// TIA Portal V20 export
// export: Created 2025-12-01T14:57:11.4895268Z, ExportSetting None, DisplayName Totally Integrated Automation Portal, DisplayVersion V20 Update 3, DisplayName TIA Portal Openness, DisplayVersion V20 Update 3, DisplayName TIA Portal Version Control Interface, DisplayVersion V20 Update 3, DisplayName STEP 7 Professional, DisplayVersion V20 Update 3, DisplayName STEP 7 Safety, DisplayVersion V20 Update 2, DisplayName WinCC Basic/Comfort/Advanced, DisplayVersion V20 Update 3, DisplayName WinCC Professional, DisplayVersion V20 Update 3, DisplayName WinCC Unified, DisplayVersion V20 Update 3
FUNCTION "FC741_GestorDispositivoCBOX" : Void   // FC741, LAD
{ S7_Optimized_Access := 'FALSE' }
// stored: AutoNumber false, SetENOAutomatically false
   VAR_INPUT
      NumCBOX : UInt;   // Numero de VTDC a Gestionar
   END_VAR
   VAR_TEMP
      RecProtocoloDispositivo : "UDT_ProtocoloRecDispositivo";   // Protocolo De Ordenes
      EmiProtocoloDispositivo : "UDT_ProtocoloEmiDispositivo";   // Protocolo De Emisiones
      P_RecProtocolo : DWord;   // Puntero a la Variable Rec Protocolo
      P_EmiProtocolo : DWord;   // Puntero a la Variable Emi Protocolo
      P_Eventos : DWord;   // Eventos - Puntero al DB de Eventos
      DBEventos : Word;   // Eventos - DB de Eventos
      NumDBEventos : UInt;   // Eventos - DB de Eventos
      MaxBytesDeEventos : UInt;   // Eventos - Maximo Bytes en el DB de Eventos
      NumBytes : UInt;   // Eventos - Numero de Bytes en el DB de Eventos
      Conversion : DWord;   // Eventos - Valor Etiqueta Convertido
      Valor : UDInt;   // Eventos - Valor Numerico a Convertir
      Convertir : UInt;   // Eventos - Valor Etiqueta a Convertir
      OffsetFinal : UInt;   // Eventos - Posicion Final
      OffsetInicial : UInt;   // Eventos - Posicion Inicial
      NumeroDispositivo : UInt;   // Temporal - Numero de CBOX
      P_Temporal : DWord;   // Temporal - Puntero
   END_VAR
BEGIN

NETWORK
TITLE = Inicializar
////////////////////////////////////////////////////////////////////////////////////////
////////////////////////////////////////////////////////////////////////////////////////
////////////////////////////////////////////////////////////////////////////////////////
// --- Inicializar Variables

      L     #NumCBOX;
      T     #NumeroDispositivo;


////////////////////////////////////////////////////////////////////////////////////////
////////////////////////////////////////////////////////////////////////////////////////
////////////////////////////////////////////////////////////////////////////////////////
// --- Recoger Protocolo de ORDEN del Dispositivo
      CALL  MOVE
      ( IN  := "DB841_Recepcion".DispoArmario[#NumeroDispositivo].Protocolo,
        OUT := #RecProtocoloDispositivo
      );

      L     P##RecProtocoloDispositivo;
      T     #P_RecProtocolo;

////////////////////////////////////////////////////////////////////////////////////////
////////////////////////////////////////////////////////////////////////////////////////
////////////////////////////////////////////////////////////////////////////////////////
// --- Recoger Protocolo de EMISION del Dispositivo
      CALL  MOVE
      ( IN  := "DB840_Emision".DispoArmario[#NumeroDispositivo].Protocolo,
        OUT := #EmiProtocoloDispositivo
      );

      L     P##EmiProtocoloDispositivo;
      T     #P_EmiProtocolo;

      L     "DB840_Emision".DispoArmario[#NumeroDispositivo].Error;
      T     "DB830_Dispositivos".Dispositivos[#NumeroDispositivo].ErrorReal;

      L     LW [#P_EmiProtocolo];
      L     W#16#7700;  // Solo la Parte Baja
      AW;
      SRD   8;
      T     "DB830_Dispositivos".Dispositivos[#NumeroDispositivo].StatusReal;



NETWORK
TITLE = Generacion de Ordenes
GeneradorDeOrdenes:NOP   0;

////////////////////////////////////////////////////////////////////////////////////////
////////////////////////////////////////////////////////////////////////////////////////
////////////////////////////////////////////////////////////////////////////////////////
// --- Fase 01 : Cierre de Protocolo de la ORDEN
      L     "DB830_Dispositivos".Dispositivos[#NumeroDispositivo].EstadoOrdenDispo;
      L     0;
      <>I;  // Mirar si no esta Cerrado el Protocolo ?
      JC    Cerrar_ProtocoloOrdenes;


////////////////////////////////////////////////////////////////////////////////////////
////////////////////////////////////////////////////////////////////////////////////////
////////////////////////////////////////////////////////////////////////////////////////
// --- Fase 02 : Eventos Recibidos (Distribucion)
      L     "DB830_Dispositivos".Dispositivos[#NumeroDispositivo].EstadoRecepcionEvento;
      L     0;  // Se han Recibido Eventos
      ==I;
      JC    Final_GeneradorDeOrdenes;


////////////////////////////////////////////////////////////////////////////////////////
// --- (260) Cambio de Estado sin Orden
      SET;
      SET;
      L     "DB830_Dispositivos".Dispositivos[#NumeroDispositivo].EstadoRecepcionEvento;
      L     260;
      ==I;
      JC    EventoRecibido_PeticionRefrescoDatos;


////////////////////////////////////////////////////////////////////////////////////////
// --- (261...274) - Recibido Ordenes para el Dispositivo
      SET;
      A(;
      L     "DB830_Dispositivos".Dispositivos[#NumeroDispositivo].EstadoRecepcionEvento;
      L     "Evento_DISPOSITIVO_InicioOrdenDipositivo";
      >=I;
      );
      A(;
      L     "DB830_Dispositivos".Dispositivos[#NumeroDispositivo].EstadoRecepcionEvento;
      L     "Evento_DISPOSITIVO_FinalOrdenDispositivo";
      <=I;
      );
      JC    EventoRecibido_OrdenesDelDipositivo;


////////////////////////////////////////////////////////////////////////////////////////
// --- (250) Peticion de Refesco de Datos del Dispositivo
      SET;
      L     "DB830_Dispositivos".Dispositivos[#NumeroDispositivo].EstadoRecepcionEvento;
      L     "Evento_DISPOSITIVO_PeticionEstadoActual";
      ==I;
      JC    EventoRecibido_PeticionRefrescoDatos;


////////////////////////////////////////////////////////////////////////////////////////
// --- No existe este Evento Programado
      L     0;  // Eliminar Evento
      T     "DB830_Dispositivos".Dispositivos[#NumeroDispositivo].EstadoRecepcionEvento;


////////////////////////////////////////////////////////////////////////////////////////
////////////////////////////////////////////////////////////////////////////////////////
////////////////////////////////////////////////////////////////////////////////////////
// --- Fase Final - No hay que hacer mas en la Generacion de Ordenes
//                  Seguir con el Generador de Emisiones
Final_GeneradorDeOrdenes:NOP   0;
      JU    GeneradorDeEmisiones;



NETWORK
TITLE = ---- Cierre del Protocolo de Ordenes del Dispositivo
Cerrar_ProtocoloOrdenes:NOP   0;

////////////////////////////////////////////////////////////////////////////////////////
////////////////////////////////////////////////////////////////////////////////////////
////////////////////////////////////////////////////////////////////////////////////////
// --- Distribuir dependiendo de la Fase del Protocolo de ORDEN

      L     "DB830_Dispositivos".Dispositivos[#NumeroDispositivo].EstadoOrdenDispo;
      L     1;
      ==I;
      JC    EnFase_01_ProtocoloOrdenes;
      JU    EnFase_02_ProtocoloOrdenes;


////////////////////////////////////////////////////////////////////////////////////////
////////////////////////////////////////////////////////////////////////////////////////
////////////////////////////////////////////////////////////////////////////////////////
// --- En Fase 01 : Esperando que se Desactive RecepOK del Dispositivo
EnFase_01_ProtocoloOrdenes:NOP   0;
      SET;  // DesActivado la RecepOK ?
      A     "DB840_Emision".DispoArmario[#NumeroDispositivo].Protocolo.RecepOK;
      JC    FinCierre_ProtocoloOrdenes;

// --- Finalizado el Protocolo
      L     0;
      T     "DB830_Dispositivos".Dispositivos[#NumeroDispositivo].EstadoOrdenDispo;
      JU    FinCierre_ProtocoloOrdenes;


////////////////////////////////////////////////////////////////////////////////////////
////////////////////////////////////////////////////////////////////////////////////////
////////////////////////////////////////////////////////////////////////////////////////
// --- Esperando que se active RecepOK del Dispositivo
EnFase_02_ProtocoloOrdenes:NOP   0;
      SET;  // DesActivado la RecepOK ?
      AN    "DB840_Emision".DispoArmario[#NumeroDispositivo].Protocolo.RecepOK;
      JC    FinCierre_ProtocoloOrdenes;

// --- Fase 01 del Protocolo
      L     1;
      T     "DB830_Dispositivos".Dispositivos[#NumeroDispositivo].EstadoOrdenDispo;

      L     LW [#P_RecProtocolo];
      L     W#16#80;
      AW;  // Desactivo la Orden enviada
      T     LW [#P_RecProtocolo];

      CALL  MOVE
      ( IN  := #RecProtocoloDispositivo,
        OUT := "DB841_Recepcion".DispoArmario[#NumeroDispositivo].Protocolo
      );

      L     0;  // Borrar Variables Auxiliares
      T     "DB841_Recepcion".DispoArmario[#NumeroDispositivo].Auxiliar_01;
      T     "DB841_Recepcion".DispoArmario[#NumeroDispositivo].Auxiliar_02;
      T     "DB841_Recepcion".DispoArmario[#NumeroDispositivo].Auxiliar_03;
      T     "DB841_Recepcion".DispoArmario[#NumeroDispositivo].ORDE;

      JU    FinCierre_ProtocoloOrdenes;


////////////////////////////////////////////////////////////////////////////////////////
////////////////////////////////////////////////////////////////////////////////////////
////////////////////////////////////////////////////////////////////////////////////////
FinCierre_ProtocoloOrdenes:NOP   0;
      JU    Final_GeneradorDeOrdenes;



NETWORK
TITLE = ---- (261...274) Recibido Ordenes para el Dipositivo
EventoRecibido_OrdenesDelDipositivo:NOP   0;

////////////////////////////////////////////////////////////////////////////////////////
////////////////////////////////////////////////////////////////////////////////////////
////////////////////////////////////////////////////////////////////////////////////////
// --- (261...274) Recibido Ordenes para el Dipositivo
      L     "DB830_Dispositivos".Dispositivos[#NumeroDispositivo].EstadoRecepcionEvento;
      L     260;
      -I;  // Numero de Bit a Activar
      L     #P_RecProtocolo;
      +D;  // Direccion del Bit a Activar
      T     #P_Temporal;

////////////////////////////////////////////////////////////////////////////////////////
// --- Activar Orden Recibida (Nuevo Estado)

      SET;  // Poner a '1' el bit de la orden
      S     L [#P_Temporal];  // Orden del PLC calculada

      CALL  MOVE
      ( IN  := #RecProtocoloDispositivo,
        OUT := "DB841_Recepcion".DispoArmario[#NumeroDispositivo].Protocolo
      );


////////////////////////////////////////////////////////////////////////////////////////
// --- Darlo por tratado y Activar Protocolo
      L     2;  // Fase 2 - Esperando que active el RecepOK
      T     "DB830_Dispositivos".Dispositivos[#NumeroDispositivo].EstadoOrdenDispo;
      L     0;  // Darlo por tratado
      T     "DB830_Dispositivos".Dispositivos[#NumeroDispositivo].EstadoRecepcionEvento;


////////////////////////////////////////////////////////////////////////////////////////
// --- Final del Evento
      JU    Final_GeneradorDeOrdenes;



NETWORK
TITLE = ---- (250 ) Peticion de Refresco de Datos del Dispositivo
EventoRecibido_PeticionRefrescoDatos:NOP   0;

////////////////////////////////////////////////////////////////////////////////////////
////////////////////////////////////////////////////////////////////////////////////////
////////////////////////////////////////////////////////////////////////////////////////
// --- 250 -  Recibido Evento de Refresco de Datos para el Dispositivo
      L     "DB830_Dispositivos".Dispositivos[#NumeroDispositivo].EstadoEmisionEvento;
      L     0;
      <>I;
      JC    Final_GeneradorDeOrdenes;


// --- (160) Refresco de datos del dispositivo
      L     "Evento_DISPOSITIVO_EstadoActual";
      T     "DB830_Dispositivos".Dispositivos[#NumeroDispositivo].EstadoEmisionEvento;

      L     0;  // Darlo por tratado
      T     "DB830_Dispositivos".Dispositivos[#NumeroDispositivo].EstadoRecepcionEvento;


////////////////////////////////////////////////////////////////////////////////////////
// --- Final del Evento
      JU    Final_GeneradorDeOrdenes;



NETWORK
TITLE = Generacion de Emisiones
GeneradorDeEmisiones:NOP   0;

////////////////////////////////////////////////////////////////////////////////////////
////////////////////////////////////////////////////////////////////////////////////////
////////////////////////////////////////////////////////////////////////////////////////
// --- Fase 01 : Cierre de Protocolo de la ORDEN
      L     "DB830_Dispositivos".Dispositivos[#NumeroDispositivo].EstadoPresenciaDispo;
      L     0;
      <>I;  // Mirar si no esta Cerrado el Protocolo ?
      JC    Cerrar_ProtocoloEmision;


////////////////////////////////////////////////////////////////////////////////////////
////////////////////////////////////////////////////////////////////////////////////////
////////////////////////////////////////////////////////////////////////////////////////
// --- Fase 02 : Comprobar si se puede Emitir Eventos
      L     "DB830_Dispositivos".Dispositivos[#NumeroDispositivo].EstadoEmisionEvento;
      L     0;
      <>I;
      JC    Final_GeneradorDeEmisiones;


////////////////////////////////////////////////////////////////////////////////////////
////////////////////////////////////////////////////////////////////////////////////////
////////////////////////////////////////////////////////////////////////////////////////
// --- Fase 03 : Tratar las Presencias (Dispositivos)
      L     LW [#P_EmiProtocolo];
      L     W#16#7F;  // Solo la Parte Alta
      AW;
      L     0;  // Mirar si se altivado algo ?
      <>I;
      JC    Tratar_PresenciaDeDipositivos;


////////////////////////////////////////////////////////////////////////////////////////
////////////////////////////////////////////////////////////////////////////////////////
////////////////////////////////////////////////////////////////////////////////////////
// --- Fase 04 : Tratar el Estado General
      SET;
      L     "DB830_Dispositivos".Dispositivos[#NumeroDispositivo].EstadoGeneralEvento;
      L     0;  // No hay nada, Petición de Evento Pendiente
      <>I;
      JC    Tratar_EventoGeneralDispositivo;


////////////////////////////////////////////////////////////////////////////////////////
////////////////////////////////////////////////////////////////////////////////////////
////////////////////////////////////////////////////////////////////////////////////////
// --- Fase 06 : Existe Cambio de Estado del Dispositivo
      L     "DB830_Dispositivos".Dispositivos[#NumeroDispositivo].StatusReal;
      L     0;
      ==I;
      JC    Final_GeneradorDeEmisiones;


// --- Es Dispositivo ha cambiado de Estado
      L     "DB830_Dispositivos".Dispositivos[#NumeroDispositivo].StatusReal;
      L     "DB830_Dispositivos".Dispositivos[#NumeroDispositivo].StatusActual;
      ==I;
      JC    Final_GeneradorDeEmisiones;


// --- Esta Activo el JDT
      SET;  // JDT 01 ???
      AN    "DB855_DefinicionDispositivos".Dispositivos[#NumeroDispositivo].EventosDelJdT02;
      AN    "DB801_JDT01StatusCOM".EnlaceCP_OK;
      JC    Final_GeneradorDeEmisiones;

      SET;  // JDT 02 ???
      A     "DB855_DefinicionDispositivos".Dispositivos[#NumeroDispositivo].EventosDelJdT02;
      AN    "DB701_JDT02StatusCOM".EnlaceCP_OK;
      JC    Final_GeneradorDeEmisiones;

      JU    Tratar_CambioEstadoDeDispositivo;


////////////////////////////////////////////////////////////////////////////////////////
////////////////////////////////////////////////////////////////////////////////////////
////////////////////////////////////////////////////////////////////////////////////////
// --- Fase Final - No hay que hacer mas en la Generacion de Emisiones
//                  Seguir con el Generador de Eventos
Final_GeneradorDeEmisiones:NOP   0;
      JU    GeneradorDeEventos;



NETWORK
TITLE = ---- Cierre del Protocolo de Emisiones del Dispositivo
Cerrar_ProtocoloEmision:NOP   0;

////////////////////////////////////////////////////////////////////////////////////////
////////////////////////////////////////////////////////////////////////////////////////
////////////////////////////////////////////////////////////////////////////////////////
// --- Esta en Fase 1 - Esperando que se desactive Emision del Dispositivo
      L     LW [#P_EmiProtocolo];
      L     W#16#7F;  // Solo la Parte Alta
      AW;
      L     0;  // Mirar si se altivado algo ?
      <>I;
      JC    FinCierre_ProtocoloEmisiones;


////////////////////////////////////////////////////////////////////////////////////////
// --- Finalizado el Protocolo
      SET;  // DesActivar - EmiOK del dispositivo
      R     "DB841_Recepcion".DispoArmario[#NumeroDispositivo].Protocolo.EmiOK;

      L     0;  // Pasar a Fase 0, Acabado el Protocolo
      T     "DB830_Dispositivos".Dispositivos[#NumeroDispositivo].EstadoPresenciaDispo;
      JU    FinCierre_ProtocoloEmisiones;


////////////////////////////////////////////////////////////////////////////////////////
////////////////////////////////////////////////////////////////////////////////////////
////////////////////////////////////////////////////////////////////////////////////////
FinCierre_ProtocoloEmisiones:NOP   0;
      JU    Final_GeneradorDeEmisiones;



NETWORK
TITLE = ---- Tratar --> Eventos de las Presencias (Dispositivos)
Tratar_PresenciaDeDipositivos:NOP   0;

/////////////////////////////////////////////////////////////////////////
/////////////////////////////////////////////////////////////////////////
/////////////////////////////////////////////////////////////////////////
// --- Distribucion por las Presencias (Generar Evento correspondiente)

      SET;  // Evento de Fin de Reset OK
      A     "DB840_Emision".DispoArmario[#NumeroDispositivo].Protocolo.ResetOK;
      JC    FinResetOK_PresenciaDeDipositivos;
      SET;  // Evento de Fin de Reset NOK
      A     "DB840_Emision".DispoArmario[#NumeroDispositivo].Protocolo.ResetNOK;
      JC    FinResetNOK_PresenciaDeDipositivos;

      SET;  // Evento de Fin de Paro Blando OK
      A     "DB840_Emision".DispoArmario[#NumeroDispositivo].Protocolo.ParoBlandoOK;
      JC    FinParoBlandoOK_PresenciaDeDipositivos;
      SET;  // Evento de Fin de Paro Blando NOK
      A     "DB840_Emision".DispoArmario[#NumeroDispositivo].Protocolo.ParoBlandoNOK;
      JC    FinParoBlandoNOK_PresenciaDeDipositivos;


/////////////////////////////////////////////////////////////////////////
/////////////////////////////////////////////////////////////////////////
/////////////////////////////////////////////////////////////////////////
// --- No hay mas tipos de presencias programadas - Cerrar el protocolo
      SET;  // Activar - EmiOK del dispositivo
      S     "DB841_Recepcion".DispoArmario[#NumeroDispositivo].Protocolo.EmiOK;

      L     1;  // Pasar a Fase 1, Empieza el Protocolo
      T     "DB830_Dispositivos".Dispositivos[#NumeroDispositivo].EstadoPresenciaDispo;
      JU    Final_GeneradorDeEmisiones;



NETWORK
TITLE = ---- Evento de las Presencia Dispositivo --> (151) Reset OK del Dispositivo
FinResetOK_PresenciaDeDipositivos:NOP   0;

/////////////////////////////////////////////////////////////////////////
/////////////////////////////////////////////////////////////////////////
/////////////////////////////////////////////////////////////////////////
// --- Generar Evento de Fin de Reset OK
      L     "Evento_DISPOSITIVO_FinReset_OK";  // 151 - Reset OK del Dispositivo
      T     "DB830_Dispositivos".Dispositivos[#NumeroDispositivo].EstadoEmisionEvento;

      SET;  // Activar - EmiOK del dispositivo
      S     "DB841_Recepcion".DispoArmario[#NumeroDispositivo].Protocolo.EmiOK;

      L     1;  // Pasar a Fase 1, Empieza el Protocolo
      T     "DB830_Dispositivos".Dispositivos[#NumeroDispositivo].EstadoPresenciaDispo;
      JU    Final_GeneradorDeEmisiones;



NETWORK
TITLE = ---- Evento de las Presencia Dispositivo --> (152) Reset NOK del Dispositivo
FinResetNOK_PresenciaDeDipositivos:NOP   0;

/////////////////////////////////////////////////////////////////////////
/////////////////////////////////////////////////////////////////////////
/////////////////////////////////////////////////////////////////////////
// --- Generar Evento de Fin de Reset NOK
      L     "Evento_DISPOSITIVO_FinReset_NOK";  // 152 - Reset NOK del Dispositivo
      T     "DB830_Dispositivos".Dispositivos[#NumeroDispositivo].EstadoEmisionEvento;

      SET;  // Activar - EmiOK del dispositivo
      S     "DB841_Recepcion".DispoArmario[#NumeroDispositivo].Protocolo.EmiOK;

      L     1;  // Pasar a Fase 1, Empieza el Protocolo
      T     "DB830_Dispositivos".Dispositivos[#NumeroDispositivo].EstadoPresenciaDispo;
      JU    Final_GeneradorDeEmisiones;



NETWORK
TITLE = ---- Evento de las Presencia Dispositivo --> (153) Paro Blando OK del Dispositivo
FinParoBlandoOK_PresenciaDeDipositivos:NOP   0;

/////////////////////////////////////////////////////////////////////////
/////////////////////////////////////////////////////////////////////////
/////////////////////////////////////////////////////////////////////////
// --- Generar Evento de Fin de Paro Blando OK
      L     "Evento_DISPOSITIVO_FinParoBlando_OK";  // 153 - Paro Blando OK del Dispositivo
      T     "DB830_Dispositivos".Dispositivos[#NumeroDispositivo].EstadoEmisionEvento;

      SET;  // Activar - EmiOK del dispositivo
      S     "DB841_Recepcion".DispoArmario[#NumeroDispositivo].Protocolo.EmiOK;

      L     1;  // Pasar a Fase 1, Empieza el Protocolo
      T     "DB830_Dispositivos".Dispositivos[#NumeroDispositivo].EstadoPresenciaDispo;
      JU    Final_GeneradorDeEmisiones;



NETWORK
TITLE = ---- Evento de las Presencia Dispositivo --> (154) Paro Blando NOK del Dispositivo
FinParoBlandoNOK_PresenciaDeDipositivos:NOP   0;

/////////////////////////////////////////////////////////////////////////
/////////////////////////////////////////////////////////////////////////
/////////////////////////////////////////////////////////////////////////
// --- Generar Evento de Fin de Paro Blando NOK
      L     "Evento_DISPOSITIVO_FinParoBlando_NOK";  // 154 - Paro Blando NOK del Dispositivo
      T     "DB830_Dispositivos".Dispositivos[#NumeroDispositivo].EstadoEmisionEvento;

      SET;  // Activar - EmiOK del dispositivo
      S     "DB841_Recepcion".DispoArmario[#NumeroDispositivo].Protocolo.EmiOK;

      L     1;  // Pasar a Fase 1, Empieza el Protocolo
      T     "DB830_Dispositivos".Dispositivos[#NumeroDispositivo].EstadoPresenciaDispo;
      JU    Final_GeneradorDeEmisiones;



NETWORK
TITLE = ---- Tratar ---> Eventos Generales de los Dispositivos
Tratar_EventoGeneralDispositivo:NOP   0;

////////////////////////////////////////////////////////////////////////////////////////
////////////////////////////////////////////////////////////////////////////////////////
////////////////////////////////////////////////////////////////////////////////////////
// --- Distribucion del Evento General del Dispositivo
      L     "DB830_Dispositivos".Dispositivos[#NumeroDispositivo].EstadoGeneralEvento;
      L     25;  // Peticion de Refesco de Datos
      ==I;
      JC    RefrescoDatos_EventoGeneralDispositivo;

// --- No hay más programados
      L     0;  // Darlo por tratado
      T     "DB830_Dispositivos".Dispositivos[#NumeroDispositivo].EstadoGeneralEvento;

      JU    Final_GeneradorDeEmisiones;



NETWORK
TITLE = ---- Evento General Dipositivo --> (160) Refesco de Estado Del Dispositivo
RefrescoDatos_EventoGeneralDispositivo:NOP   0;

////////////////////////////////////////////////////////////////////////////////////////
////////////////////////////////////////////////////////////////////////////////////////
////////////////////////////////////////////////////////////////////////////////////////
// --- Generar Evento de Refesco de Datos del Dispositivo

      L     "DB830_Dispositivos".Dispositivos[#NumeroDispositivo].StatusReal;
      T     "DB830_Dispositivos".Dispositivos[#NumeroDispositivo].StatusActual;
      L     "DB830_Dispositivos".Dispositivos[#NumeroDispositivo].ErrorReal;
      T     "DB830_Dispositivos".Dispositivos[#NumeroDispositivo].ErrorActual;

      L     0;  // EstadoGeneral - Dar por Tratado
      T     "DB830_Dispositivos".Dispositivos[#NumeroDispositivo].EstadoGeneralEvento;

// --- Comprobar que hay algo para generar
      L     "DB830_Dispositivos".Dispositivos[#NumeroDispositivo].StatusActual;
      L     0;
      ==I;
      JC    Final_GeneradorDeEmisiones;

      L     "Evento_DISPOSITIVO_EstadoActual";  // 160 - Refresco de Estado del Dispositivo
      T     "DB830_Dispositivos".Dispositivos[#NumeroDispositivo].EstadoEmisionEvento;
      JU    Final_GeneradorDeEmisiones;



NETWORK
TITLE = ---- Tratar ---> Cambio de Estado del Dispositivo
Tratar_CambioEstadoDeDispositivo:NOP   0;

////////////////////////////////////////////////////////////////////////////////////////
////////////////////////////////////////////////////////////////////////////////////////
////////////////////////////////////////////////////////////////////////////////////////
// --- Activar Evento (160) - Refresco del Estado del Dispositivo
      L     "DB830_Dispositivos".Dispositivos[#NumeroDispositivo].StatusReal;
      T     "DB830_Dispositivos".Dispositivos[#NumeroDispositivo].StatusActual;
      L     "DB830_Dispositivos".Dispositivos[#NumeroDispositivo].ErrorReal;
      T     "DB830_Dispositivos".Dispositivos[#NumeroDispositivo].ErrorActual;

      L     "Evento_DISPOSITIVO_EstadoActual";  // 160 - Refresco de Estado del Dispositivo
      T     "DB830_Dispositivos".Dispositivos[#NumeroDispositivo].EstadoEmisionEvento;

      JU    Final_GeneradorDeEmisiones;



NETWORK
TITLE = Generacion de Eventos
GeneradorDeEventos:NOP   0;

////////////////////////////////////////////////////////////////////////////////////////
////////////////////////////////////////////////////////////////////////////////////////
////////////////////////////////////////////////////////////////////////////////////////
// --- Existen Eventos a Emitir
      L     "DB830_Dispositivos".Dispositivos[#NumeroDispositivo].EstadoEmisionEvento;
      L     0;
      ==I;
      JC    Final_GeneradorDeEventos;


////////////////////////////////////////////////////////////////////////////////////////
////////////////////////////////////////////////////////////////////////////////////////
////////////////////////////////////////////////////////////////////////////////////////
// --- Variables para la Emision de Eventos (Depende del JDT)
      L     "JDT1_NDB_EventosEmi";
      T     #DBEventos;
      T     #NumDBEventos;
      L     "JDT1_MaxBytes";
      T     #MaxBytesDeEventos;

      SET;
      AN    "DB855_DefinicionDispositivos".Dispositivos[#NumeroDispositivo].EventosDelJdT02;
      JN    NoEsDispositivo_JDT02;

      L     "JDT2_NDB_EventosEmi";
      T     #DBEventos;
      T     #NumDBEventos;
      L     "JDT2_MaxBytes";
      T     #MaxBytesDeEventos;

NoEsDispositivo_JDT02:NOP   0;


////////////////////////////////////////////////////////////////////////////////////////
////////////////////////////////////////////////////////////////////////////////////////
////////////////////////////////////////////////////////////////////////////////////////
// --- Hay espacio para la Emision de Eventos
      L     0;
      T     #NumBytes;  // Inicializo el numero de Bytes
      LAR2;  // Inicializo el puntero de Eventos Generados

////////////////////////////////////////////////////////////////////////////////////////
// --- Calcula el tamaño de bytes que hay en el DB Eventos Generados

      OPN   DB [#DBEventos];
InicioBucleBusquedaFin_BufferEventos:NOP   0;
      L     DBB [AR2, P#0.0];
      L     0;
      ==I;  // Buscamos el final del DB = 0
      JC    FinalBucleBusquedaFin_BufferEventos;

      +AR2  P#1.0;
      JU    InicioBucleBusquedaFin_BufferEventos;

FinalBucleBusquedaFin_BufferEventos:NOP   0;
      TAR2;  // Guardo el puntero
      T     #P_Eventos;  // Sacamos el NumBytes Escritos
      SRD   3;
      T     #NumBytes;

////////////////////////////////////////////////////////////////////////////////////////
// --- Comprobamos si hay sitio para mas Eventos

      L     #NumBytes;  // Miramos si hay sitio
      L     #MaxBytesDeEventos;  // Max. que se pueden emitir, parametro
      >I;  // No se pueden generar más eventos
      JC    Final_GeneradorDeEventos;


////////////////////////////////////////////////////////////////////////////////////////
////////////////////////////////////////////////////////////////////////////////////////
////////////////////////////////////////////////////////////////////////////////////////
// --- Distribuir Segun Evento a Emitir


////////////////////////////////////////////////////////////////////////////////////////
// --- Estado del Dispositivo
      L     "DB830_Dispositivos".Dispositivos[#NumeroDispositivo].EstadoEmisionEvento;
      L     "Evento_DISPOSITIVO_EstadoActual";
      ==I;
      JC    GenerarEvento_EstadoDispositivo;


////////////////////////////////////////////////////////////////////////////////////////
// --- Fin de Reset
      L     "DB830_Dispositivos".Dispositivos[#NumeroDispositivo].EstadoEmisionEvento;
      L     "Evento_DISPOSITIVO_FinReset_OK";
      ==I;
      JC    GenerarEvento_FinResetProcesoDispositivo;
      L     "DB830_Dispositivos".Dispositivos[#NumeroDispositivo].EstadoEmisionEvento;
      L     "Evento_DISPOSITIVO_FinReset_NOK";
      ==I;
      JC    GenerarEvento_FinResetProcesoDispositivo;


////////////////////////////////////////////////////////////////////////////////////////
// --- Fin de Paro Blando
      L     "DB830_Dispositivos".Dispositivos[#NumeroDispositivo].EstadoEmisionEvento;
      L     "Evento_DISPOSITIVO_FinParoBlando_OK";
      ==I;
      JC    GenerarEvento_FinParoBlandoProcesoDispositivo;
      L     "DB830_Dispositivos".Dispositivos[#NumeroDispositivo].EstadoEmisionEvento;
      L     "Evento_DISPOSITIVO_FinParoBlando_NOK";
      ==I;
      JC    GenerarEvento_FinParoBlandoProcesoDispositivo;


////////////////////////////////////////////////////////////////////////////////////////
////////////////////////////////////////////////////////////////////////////////////////
////////////////////////////////////////////////////////////////////////////////////////
// --- Evento a Emitir NO VALIDO
      L     0;
      T     "DB830_Dispositivos".Dispositivos[#NumeroDispositivo].EstadoEmisionEvento;
      JU    Final_GeneradorDeEventos;


////////////////////////////////////////////////////////////////////////////////////////
////////////////////////////////////////////////////////////////////////////////////////
////////////////////////////////////////////////////////////////////////////////////////
// --- Fase Final - No hay que hacer mas en la Generacion de Eventos
Final_GeneradorDeEventos:NOP   0;
      BE;  // Finalizar Funcion



NETWORK
TITLE = ---- Generar el Evento STAT --> Estado del Dispositivo
GenerarEvento_EstadoDispositivo:NOP   0;

////////////////////////////////////////////////////////////////////////////////////////
////////////////////////////////////////////////////////////////////////////////////////
////////////////////////////////////////////////////////////////////////////////////////
// --- Evento de Dispositivo - Estado de Dispositivo - STAT
      LAR2  #P_Eventos;  // Puntero al DB de Eventos Generados

// --- Separacion entre Eventos a Generar
      L     #P_Eventos;  // Mirar si es el primer evento de la lista
      L     0;  // Es el primero ?
      ==I;
      JC    InicioBuffer_EventoSTAT_EstadoDispositivo;

      OPN   DB [#DBEventos];
      L     ',';  // Separador entre eventos ','
      T     DBB [AR2, P#0.0];
      +AR2  P#1.0;

InicioBuffer_EventoSTAT_EstadoDispositivo:NOP   0;


////////////////////////////////////////////////////////////////////////////////////////
////////////////////////////////////////////////////////////////////////////////////////
////////////////////////////////////////////////////////////////////////////////////////
// --- Inicio de Evento
      OPN   DB [#DBEventos];  // DB de Eventos Generados (A Emitir)
      L     '{';  // Inicio de Evento '{'
      T     DBB [AR2, P#0.0];
      +AR2  P#1.0;

      L     'STAT';  // Evento 'STAT'
      T     DBD [AR2, P#0.0];
      +AR2  P#4.0;


////////////////////////////////////////////////////////////////////////////////////////
// --- Atributo Tipo '[TIPO]'

      OPN   DB [#DBEventos];
      L     '[';
      T     DBB [AR2, P#0.0];
      L     'TIPO';
      T     DBD [AR2, P#1.0];
      L     ']';
      T     DBB [AR2, P#5.0];
      +AR2  P#6.0;

      L     'CBOX';
      T     DBD [AR2, P#0.0];
      +AR2  P#4.0;

////////////////////////////////////////////////////////////////////////////////////////
// --- Atributo Numero de Dispositivo '[NUME]'
      OPN   DB [#DBEventos];
      L     '[';
      T     DBB [AR2, P#0.0];
      L     'NUME';
      T     DBD [AR2, P#1.0];
      L     ']';
      T     DBB [AR2, P#5.0];
      +AR2  P#6.0;

      L     "CTE_OffsetCCPIF";
      L     1;
      +I;
      L     100;
      *I;
      L     #NumeroDispositivo;  // Numero de Dispo
      +I;
      T     #Valor;

// --- Convertir Valor a ASCII - Numero de Dispositivo
      TAR2;
      SRD   3;
      T     #OffsetInicial;  // Miro que offset tiene la String

      CALL  "FC893_Obtener_StringDelAtributo"
      ( DB_String := #NumDBEventos,
        OffsetIni := #OffsetInicial,
        Valor     := #Valor,
        OffsetFin := #OffsetFinal
      );  // Llamo a ObtenerStrinAtributo

      L     #OffsetFinal;
      SLD   3;
      LAR2;  // Recupero que offset tiene la String


////////////////////////////////////////////////////////////////////////////////////////
// --- Atributo Numero de Dispositivo '[NUES]'
      OPN   DB [#DBEventos];
      L     '[';
      T     DBB [AR2, P#0.0];
      L     'NUES';
      T     DBD [AR2, P#1.0];
      L     ']';
      T     DBB [AR2, P#5.0];
      +AR2  P#6.0;

      L     "DB830_Dispositivos".Dispositivos[#NumeroDispositivo].StatusActual;
      L     W#16#F;  // Solo la parte Estado
      AW;
      T     #Convertir;

      CALL  "FC895_Obtener_EtiquetaDeValor"
      ( ValorEvento    := #Convertir,
        EtiquetaEvento := #Conversion
      );

      OPN   DB [#DBEventos];
      L     #Conversion;
      T     DBD [AR2, P#0.0];
      +AR2  P#4.0;


////////////////////////////////////////////////////////////////////////////////////////
// --- Atributo Numero de Dispositivo '[LLAV]'
      OPN   DB [#DBEventos];
      L     '[';  // Evento -
      T     DBB [AR2, P#0.0];
      L     'LLAV';
      T     DBD [AR2, P#1.0];
      L     ']';
      T     DBB [AR2, P#5.0];
      +AR2  P#6.0;

      L     "DB830_Dispositivos".Dispositivos[#NumeroDispositivo].StatusActual;
      L     W#16#F0;  // Solo la parte Llave
      AW;
      SRD   4;
      L     10;
      +I;
      T     #Convertir;

      T     #Convertir;
      CALL  "FC895_Obtener_EtiquetaDeValor"
      ( ValorEvento    := #Convertir,
        EtiquetaEvento := #Conversion
      );

      OPN   DB [#DBEventos];
      L     #Conversion;
      T     DBD [AR2, P#0.0];
      +AR2  P#4.0;


////////////////////////////////////////////////////////////////////////////////////////
// --- Poner Error (Si es necesario)
      L     "DB830_Dispositivos".Dispositivos[#NumeroDispositivo].ErrorActual;
      L     0;
      ==D;
      JC    NoErrorDispositivo_STAT_EstadoDispositivo;


// --- Atributo Numero de Dispositivo '[CODE]'
      OPN   DB [#DBEventos];
      L     '[';  // Evento -
      T     DBB [AR2, P#0.0];
      L     'CODE';
      T     DBD [AR2, P#1.0];
      L     ']';
      T     DBB [AR2, P#5.0];
      +AR2  P#6.0;

      L     "DB830_Dispositivos".Dispositivos[#NumeroDispositivo].ErrorActual;
      T     #Valor;

// --- Convertir Valor a ASCII - Error
      TAR2;
      SRD   3;
      T     #OffsetInicial;  // Miro que offset tiene la String

      CALL  "FC893_Obtener_StringDelAtributo"
      ( DB_String := #NumDBEventos,
        OffsetIni := #OffsetInicial,
        Valor     := #Valor,
        OffsetFin := #OffsetFinal
      );  // Llamo a ObtenerStrinAtributo

      L     #OffsetFinal;
      SLD   3;
      LAR2;  // Recupero que offset tiene la String

NoErrorDispositivo_STAT_EstadoDispositivo:NOP   0;


////////////////////////////////////////////////////////////////////////////////////////
// --- Final del formaateo del Evento
      OPN   DB [#DBEventos];  // DB de Eventos Generados (A Emitir)
      L     '}';  // Fin de Evento '}'
      T     DBB [AR2, P#0.0];
      +AR2  P#1.0;


////////////////////////////////////////////////////////////////////////////////////////
////////////////////////////////////////////////////////////////////////////////////////
////////////////////////////////////////////////////////////////////////////////////////
// --- Dar por formateado el Evento

      L     0;  // 0 - Lo doy por tratado
      T     "DB830_Dispositivos".Dispositivos[#NumeroDispositivo].EstadoEmisionEvento;

      JU    Final_GeneradorDeEventos;



NETWORK
TITLE = ---- Generar el Evento FIN! --> Reset OK, Reset NOK
GenerarEvento_FinResetProcesoDispositivo:NOP   0;

////////////////////////////////////////////////////////////////////////////////////////
////////////////////////////////////////////////////////////////////////////////////////
////////////////////////////////////////////////////////////////////////////////////////
// --- Formateo del Evento FIN! (Fin del Proceso --> Reset y Paro Blando)
      LAR2  #P_Eventos;  // Puntero al DB de Eventos Generados

// --- Separacion entre Eventos a Generar
      L     #P_Eventos;  // Mirar si es el primer evento de la lista
      L     0;  // Es el primero ?
      ==I;
      JC    InicioBuffer_EventoFIN_FinResetProcesoDispositivo;

      OPN   DB [#DBEventos];
      L     ',';  // Separador entre eventos ','
      T     DBB [AR2, P#0.0];
      +AR2  P#1.0;

InicioBuffer_EventoFIN_FinResetProcesoDispositivo:NOP   0;


////////////////////////////////////////////////////////////////////////////////////////
////////////////////////////////////////////////////////////////////////////////////////
////////////////////////////////////////////////////////////////////////////////////////
// --- Inicio de Evento
      OPN   DB [#DBEventos];  // DB de Eventos Generados (A Emitir)
      L     '{';  // Inicio de Evento '{'
      T     DBB [AR2, P#0.0];
      +AR2  P#1.0;

      L     'FIN!';  // Evento 'FIN!'
      T     DBD [AR2, P#0.0];
      +AR2  P#4.0;


////////////////////////////////////////////////////////////////////////////////////////
// --- Atributo Tipo '[TIPO]'

      OPN   DB [#DBEventos];
      L     '[';
      T     DBB [AR2, P#0.0];
      L     'TIPO';
      T     DBD [AR2, P#1.0];
      L     ']';
      T     DBB [AR2, P#5.0];
      +AR2  P#6.0;


      L     'CBOX';
      T     DBD [AR2, P#0.0];
      +AR2  P#4.0;

////////////////////////////////////////////////////////////////////////////////////////
// --- Atributo Numero de Dispositivo '[NUME]'
      OPN   DB [#DBEventos];
      L     '[';
      T     DBB [AR2, P#0.0];
      L     'NUME';
      T     DBD [AR2, P#1.0];
      L     ']';
      T     DBB [AR2, P#5.0];
      +AR2  P#6.0;

      L     "CTE_OffsetCCPIF";
      L     1;
      +I;
      L     100;
      *I;
      L     #NumeroDispositivo;  // Numero de Dispo
      +I;
      T     #Valor;

// --- Convertir Valor a ASCII - Numero de Dispositivo
      TAR2;
      SRD   3;
      T     #OffsetInicial;  // Miro que offset tiene la String

      CALL  "FC893_Obtener_StringDelAtributo"
      ( DB_String := #NumDBEventos,
        OffsetIni := #OffsetInicial,
        Valor     := #Valor,
        OffsetFin := #OffsetFinal
      );  // Llamo a ObtenerStrinAtributo

      L     #OffsetFinal;
      SLD   3;
      LAR2;  // Recupero que offset tiene la String


////////////////////////////////////////////////////////////////////////////////////////
// --- Atributo Numero de Dispositivo '[PROC]'
      OPN   DB [#DBEventos];
      L     '[';
      T     DBB [AR2, P#0.0];
      L     'PROC';
      T     DBD [AR2, P#1.0];
      L     ']';
      T     DBB [AR2, P#5.0];
      +AR2  P#6.0;

      OPN   DB [#DBEventos];
      L     'RESE';
      T     DBD [AR2, P#0.0];
      +AR2  P#4.0;


////////////////////////////////////////////////////////////////////////////////////////
// --- Atributo Numero de Dispositivo '[RSLT]'
      OPN   DB [#DBEventos];
      L     '[';
      T     DBB [AR2, P#0.0];
      L     'RSLT';
      T     DBD [AR2, P#1.0];
      L     ']';
      T     DBB [AR2, P#5.0];
      +AR2  P#6.0;

      L     "DB830_Dispositivos".Dispositivos[#NumeroDispositivo].EstadoEmisionEvento;
      L     151;
      -I;
      L     W#16#30;  // Convertir a ASCII
      +I;
      OPN   DB [#DBEventos];
      T     DBB [AR2, P#0.0];
      +AR2  P#1.0;


////////////////////////////////////////////////////////////////////////////////////////
// --- Final del formaateo del Evento
      OPN   DB [#DBEventos];  // DB de Eventos Generados (A Emitir)
      L     '}';  // Fin de Evento '}'
      T     DBB [AR2, P#0.0];
      +AR2  P#1.0;


////////////////////////////////////////////////////////////////////////////////////////
////////////////////////////////////////////////////////////////////////////////////////
////////////////////////////////////////////////////////////////////////////////////////
// --- Dar por formateado el Evento

      L     0;  // 0 - Lo doy por tratado
      T     "DB830_Dispositivos".Dispositivos[#NumeroDispositivo].EstadoEmisionEvento;

      JU    Final_GeneradorDeEventos;




NETWORK
TITLE = ---- Generar el Evento FIN! --> ParoBlando OK ParoBlandoNOK
GenerarEvento_FinParoBlandoProcesoDispositivo:NOP   0;

////////////////////////////////////////////////////////////////////////////////////////
////////////////////////////////////////////////////////////////////////////////////////
////////////////////////////////////////////////////////////////////////////////////////
// --- Formateo del Evento FIN! (Fin del Proceso --> Reset y Paro Blando)
      LAR2  #P_Eventos;  // Puntero al DB de Eventos Generados

// --- Separacion entre Eventos a Generar
      L     #P_Eventos;  // Mirar si es el primer evento de la lista
      L     0;  // Es el primero ?
      ==I;
      JC    InicioBuffer_EventoFIN_FinParoBlandoProcesoDispositivo;

      OPN   DB [#DBEventos];
      L     ',';  // Separador entre eventos ','
      T     DBB [AR2, P#0.0];
      +AR2  P#1.0;

InicioBuffer_EventoFIN_FinParoBlandoProcesoDispositivo:NOP   0;


////////////////////////////////////////////////////////////////////////////////////////
////////////////////////////////////////////////////////////////////////////////////////
////////////////////////////////////////////////////////////////////////////////////////
// --- Inicio de Evento
      OPN   DB [#DBEventos];  // DB de Eventos Generados (A Emitir)
      L     '{';  // Inicio de Evento '{'
      T     DBB [AR2, P#0.0];
      +AR2  P#1.0;

      L     'FIN!';  // Evento 'FIN!'
      T     DBD [AR2, P#0.0];
      +AR2  P#4.0;


////////////////////////////////////////////////////////////////////////////////////////
// --- Atributo Tipo '[TIPO]'

      OPN   DB [#DBEventos];
      L     '[';
      T     DBB [AR2, P#0.0];
      L     'TIPO';
      T     DBD [AR2, P#1.0];
      L     ']';
      T     DBB [AR2, P#5.0];
      +AR2  P#6.0;


      L     'CBOX';
      T     DBD [AR2, P#0.0];
      +AR2  P#4.0;

////////////////////////////////////////////////////////////////////////////////////////
// --- Atributo Numero de Dispositivo '[NUME]'
      OPN   DB [#DBEventos];
      L     '[';
      T     DBB [AR2, P#0.0];
      L     'NUME';
      T     DBD [AR2, P#1.0];
      L     ']';
      T     DBB [AR2, P#5.0];
      +AR2  P#6.0;

      L     "CTE_OffsetCCPIF";
      L     1;
      +I;
      L     100;
      *I;
      L     #NumeroDispositivo;  // Numero de Dispo
      +I;
      T     #Valor;

// --- Convertir Valor a ASCII - Numero de Dispositivo
      TAR2;
      SRD   3;
      T     #OffsetInicial;  // Miro que offset tiene la String

      CALL  "FC893_Obtener_StringDelAtributo"
      ( DB_String := #NumDBEventos,
        OffsetIni := #OffsetInicial,
        Valor     := #Valor,
        OffsetFin := #OffsetFinal
      );  // Llamo a ObtenerStrinAtributo

      L     #OffsetFinal;
      SLD   3;
      LAR2;  // Recupero que offset tiene la String


////////////////////////////////////////////////////////////////////////////////////////
// --- Atributo Numero de Dispositivo '[PROC]'
      OPN   DB [#DBEventos];
      L     '[';
      T     DBB [AR2, P#0.0];
      L     'PROC';
      T     DBD [AR2, P#1.0];
      L     ']';
      T     DBB [AR2, P#5.0];
      +AR2  P#6.0;

      OPN   DB [#DBEventos];
      L     'BLAN';
      T     DBD [AR2, P#0.0];
      +AR2  P#4.0;


////////////////////////////////////////////////////////////////////////////////////////
// --- Atributo Numero de Dispositivo '[RSLT]'
      OPN   DB [#DBEventos];
      L     '[';
      T     DBB [AR2, P#0.0];
      L     'RSLT';
      T     DBD [AR2, P#1.0];
      L     ']';
      T     DBB [AR2, P#5.0];
      +AR2  P#6.0;

      L     "DB830_Dispositivos".Dispositivos[#NumeroDispositivo].EstadoEmisionEvento;
      L     153;
      -I;
      L     W#16#30;  // Convertir a ASCII
      +I;
      OPN   DB [#DBEventos];
      T     DBB [AR2, P#0.0];
      +AR2  P#1.0;


////////////////////////////////////////////////////////////////////////////////////////
// --- Final del formaateo del Evento
      OPN   DB [#DBEventos];  // DB de Eventos Generados (A Emitir)
      L     '}';  // Fin de Evento '}'
      T     DBB [AR2, P#0.0];
      +AR2  P#1.0;


////////////////////////////////////////////////////////////////////////////////////////
////////////////////////////////////////////////////////////////////////////////////////
////////////////////////////////////////////////////////////////////////////////////////
// --- Dar por formateado el Evento

      L     0;  // 0 - Lo doy por tratado
      T     "DB830_Dispositivos".Dispositivos[#NumeroDispositivo].EstadoEmisionEvento;

      JU    Final_GeneradorDeEventos;



END_FUNCTION
